{attribute 'GeneratedUsingTerminal: KL2212'}
{attribute addProperty BoxType "KL2212"}
{attribute addProperty Id "Channel_1AT %Q*Channel_DCF170BB0Channel_2AT %Q*Channel_DCF170BB0"}
{attribute addProperty CRC "3122143290"}
{attribute addProperty Size "0"}
TYPE KL2212_BA18203A :
STRUCT
	{attribute addProperty Name "Channel_1"}
	Channel_1 : Channel_DCF170BB;
	{attribute addProperty Name "Channel_2"}
	Channel_2 : Channel_DCF170BB;
END_STRUCT
END_TYPE

(* stored: Version 1.2.0.0, ProductVersion 3.1.4024.9
   DUT KL2212_BA18203A: Id {69988c9f-4773-49c0-bc7c-1e793661eac9} *)
